// TIA Portal V16 export
// export: Created 2023-03-29T11:04:44.9986419Z, ExportSetting WithDefaults, DisplayName Totally Integrated Automation Portal, DisplayVersion V16 Update 6, DisplayName TIA Portal Version Control Interface, DisplayVersion V16 Update 2, DisplayName TIA Portal Openness, DisplayVersion V16 Update 6, DisplayName STEP 7 Professional, DisplayVersion V16 Update 6, DisplayName STEP 7 Safety, DisplayVersion V16, DisplayName WinCC Advanced, DisplayVersion V16 Update 6
FUNCTION "Sterowniki_Z11_Z12" : Void   // FC30, LAD
TITLE = Driver napedów zasuw Z11, Z12
{ S7_Optimized_Access := 'TRUE' }
AUTHOR : rtecmer
VERSION : 0.1
// Funkcje sterujące napędami w trybie zdalnym, lokalnym
// stored: AutoNumber true, IsIECCheckEnabled false, SetENOAutomatically false, UDAEnableTagReadback false
BEGIN

REGION Network 1: Zasuwa Z11
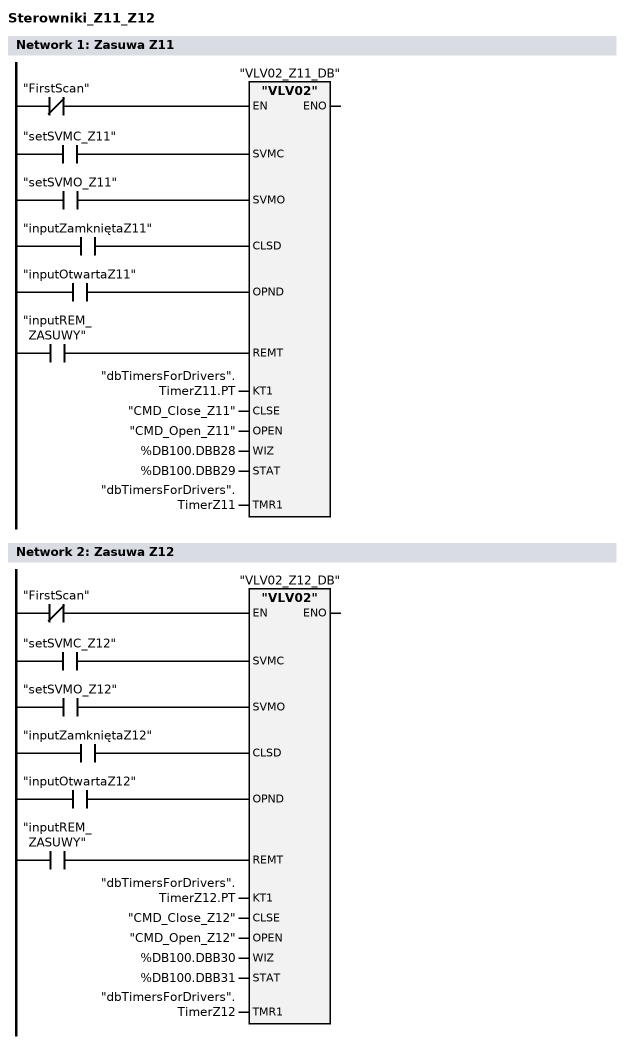
   RUNG wire#powerrail
      I_Contact( "FirstScan" )
      "VLV02_Z11_DB"(SVMC := wire#w1, SVMO := wire#w2, CLSD := wire#w3, OPND := wire#w4, REMT := wire#w5, KT1 := "dbTimersForDrivers".TimerZ11.PT, CLSE := "CMD_Close_Z11", OPEN := "CMD_Open_Z11", WIZ := %DB100.DBB28, STAT := %DB100.DBB29, TMR1 := "dbTimersForDrivers".TimerZ11)
   END_RUNG
   RUNG wire#powerrail
      Contact( "setSVMC_Z11" )
   END_RUNG wire#w1
   RUNG wire#powerrail
      Contact( "setSVMO_Z11" )
   END_RUNG wire#w2
   RUNG wire#powerrail
      Contact( "inputZamkniętaZ11" )
   END_RUNG wire#w3
   RUNG wire#powerrail
      Contact( "inputOtwartaZ11" )
   END_RUNG wire#w4
   RUNG wire#powerrail
      Contact( "inputREM_ZASUWY" )
   END_RUNG wire#w5
   // the same network as SCL:
   IF NOT "FirstScan" THEN
       "VLV02_Z11_DB"(SVMC := "setSVMC_Z11",   // "VLV02"
                      SVMO := "setSVMO_Z11",
                      CLSD := "inputZamkniętaZ11",
                      OPND := "inputOtwartaZ11",
                      REMT := "inputREM_ZASUWY",
                      KT1 := "dbTimersForDrivers".TimerZ11.PT,
                      CLSE := "CMD_Close_Z11",
                      OPEN := "CMD_Open_Z11",
                      WIZ := %DB100.DBB28,
                      STAT := %DB100.DBB29,
                      TMR1 := "dbTimersForDrivers".TimerZ11);
   END_IF;
END_REGION

REGION Network 2: Zasuwa Z12
   RUNG wire#powerrail
      I_Contact( "FirstScan" )
      "VLV02_Z12_DB"(SVMC := wire#w1, SVMO := wire#w2, CLSD := wire#w3, OPND := wire#w4, REMT := wire#w5, KT1 := "dbTimersForDrivers".TimerZ12.PT, CLSE := "CMD_Close_Z12", OPEN := "CMD_Open_Z12", WIZ := %DB100.DBB30, STAT := %DB100.DBB31, TMR1 := "dbTimersForDrivers".TimerZ12)
   END_RUNG
   RUNG wire#powerrail
      Contact( "setSVMC_Z12" )
   END_RUNG wire#w1
   RUNG wire#powerrail
      Contact( "setSVMO_Z12" )
   END_RUNG wire#w2
   RUNG wire#powerrail
      Contact( "inputZamkniętaZ12" )
   END_RUNG wire#w3
   RUNG wire#powerrail
      Contact( "inputOtwartaZ12" )
   END_RUNG wire#w4
   RUNG wire#powerrail
      Contact( "inputREM_ZASUWY" )
   END_RUNG wire#w5
   // the same network as SCL:
   IF NOT "FirstScan" THEN
       "VLV02_Z12_DB"(SVMC := "setSVMC_Z12",   // "VLV02"
                      SVMO := "setSVMO_Z12",
                      CLSD := "inputZamkniętaZ12",
                      OPND := "inputOtwartaZ12",
                      REMT := "inputREM_ZASUWY",
                      KT1 := "dbTimersForDrivers".TimerZ12.PT,
                      CLSE := "CMD_Close_Z12",
                      OPEN := "CMD_Open_Z12",
                      WIZ := %DB100.DBB30,
                      STAT := %DB100.DBB31,
                      TMR1 := "dbTimersForDrivers".TimerZ12);
   END_IF;
END_REGION
END_FUNCTION
